PROGRAM p_MPSSup
VAR
END_VAR

//currently only check the VGC before stopper 4.5, make sure to include the g_xIOState variable to ensure MPS is valid only when the bus is working
//q_xDG1_MMS01_MPSOK := i_xDG1_MMS01_OUT XOR i_xDG1_MMS01_IN;
//q_xMFX_MPSOK := g_xIOState AND vgcMXT_VGC_04.i_xOpnLS AND vgcDVD_VGC_01.i_xOpnLS AND 
//( i_xMFX_ppsStopperPos_In OR ( NOT(i_xMFX_ppsStopperPos_Out AND i_xMFX_ppsStopperPos_In) AND vgcDIA_VGC_01.i_xOpnLS AND vgcDIA_VGC_02.i_xOpnLS AND 
//									vgcDG1_VGC_01.i_xOpnLS AND vgcDG1_VGC_02.i_xOpnLS AND q_xDG1_MMS01_MPSOK AND i_xMFX_TFSmpsStatus_OK));
									
(* q_xMFX_preS45_MPSOK:= g_xIOState AND vgcMXT_VGC_04.i_xOpnLS AND vgcDVD_VGC_01.i_xOpnLS; 								
q_xDG1_MMS01_MPSOK := i_xDG1_MMS01_OUT AND NOT i_xDG1_MMS01_IN;
q_xMFX_VGC_OK      := vgcDIA_VGC_01.i_xOpnLS AND vgcDIA_VGC_02.i_xOpnLS
                       AND  vgcDG1_VGC_01.i_xOpnLS AND vgcDG1_VGC_02.i_xOpnLS;  								

q_xMFX_MPSOK := q_xMFX_VGC_OK AND q_xDG1_MMS01_MPSOK; *)

END_PROGRAM

(* stored: Version 1.1.0.1, ProductVersion 3.1.4020.12
   POU p_MPSSup: Id {606dda39-341f-4609-835a-4778708a8932}, SpecialFunc None *)
